SUBAPPLICATION Uebung_122_AX (* Übung zu ISOBUS Name *)
  (* Standard: 61499-2; Description: Copyright (c) 2023 Meisterschulen am Ostbahnhof This program and the accompanying materials are made available under the terms of the Eclipse Public License 2.0 which is available at https://www.eclipse.org/legal/epl-2.0/ SPDX-License-Identifier: EPL-2.0 *)
  (* Version 1.0, 2023-10-23, Franz Höpfinger, Meisterschulen am Ostbahnhof, initial API and implementation and/or initial documentation *)
  PACKAGE Uebungen;
  IMPORT Uebungen::const::Uebung_120_129::Filter::ADD_ALL_PASS;
  IMPORT Uebungen::const::Uebung_120_129::Filter::FLT_ALL_PASS;
  IMPORT isobus::pgn::ISOUSERHOME_e::network;
  IMPORT isobus::pgn::ISO_CAN_NODE::NODE1;
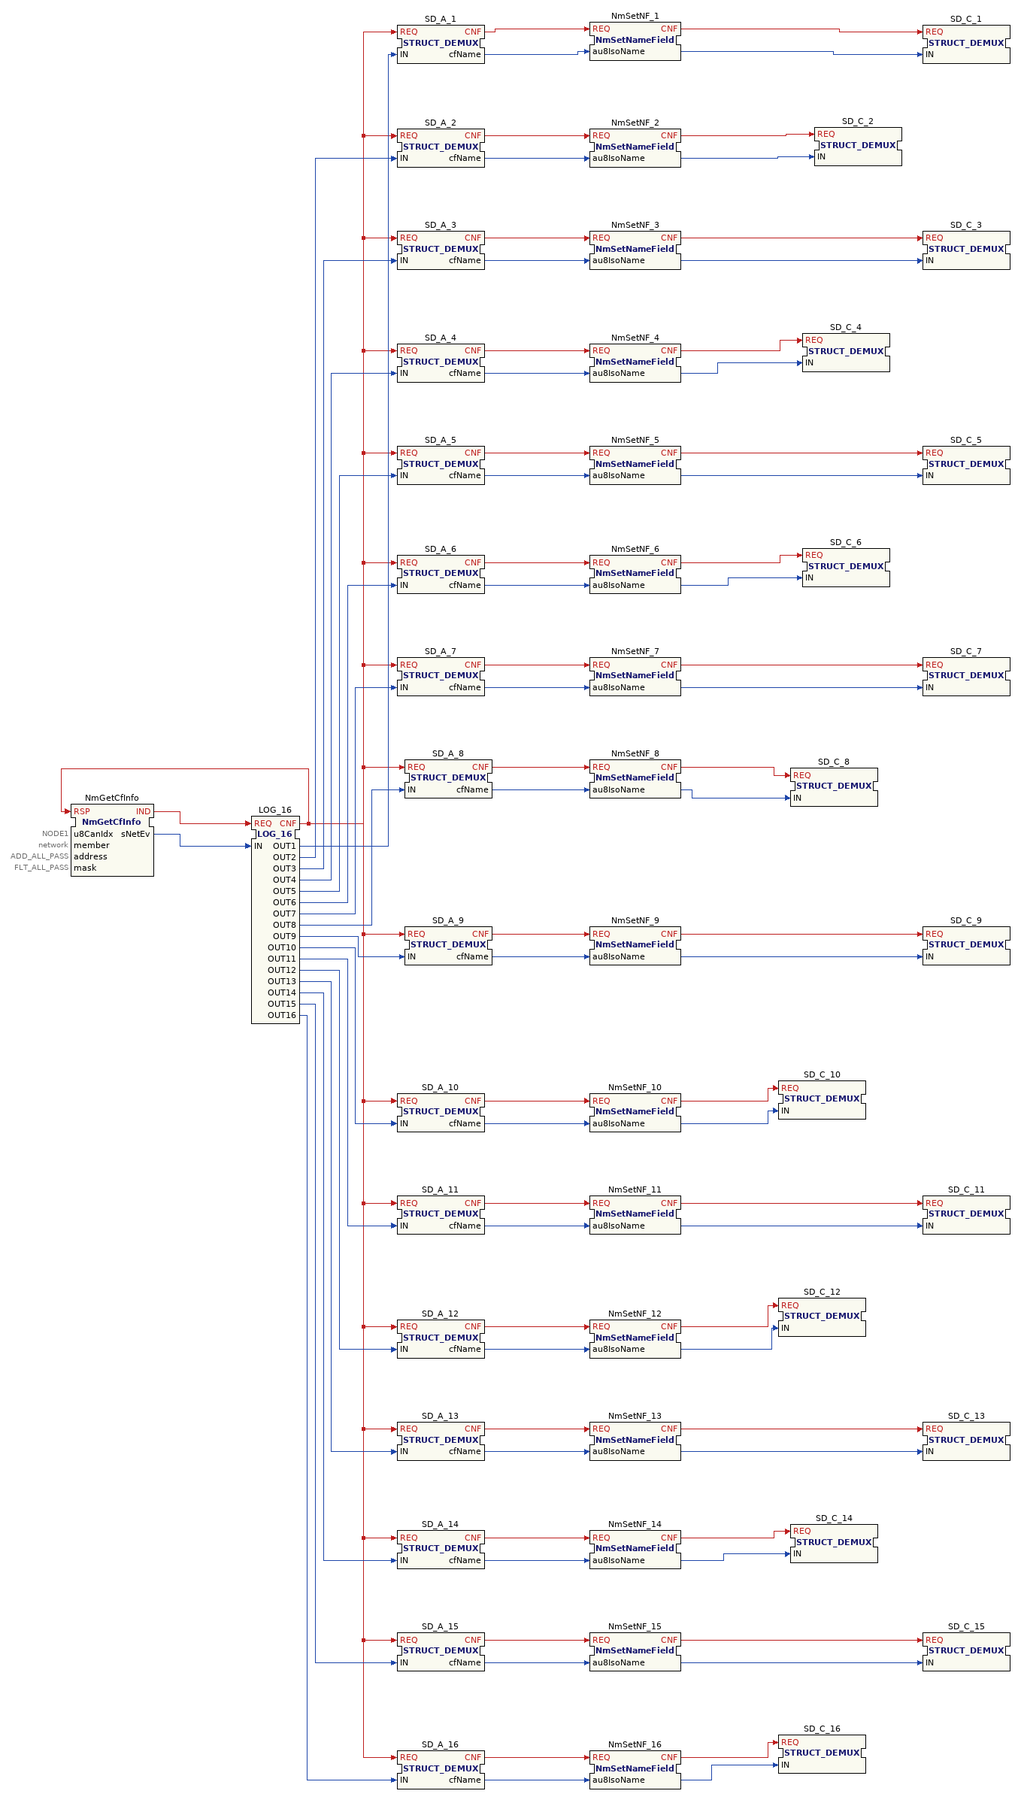
  FBS
    NmGetCfInfo : isobus::pgn::NmGetCfInfo(u8CanIdx := NODE1, member := network, address := ADD_ALL_PASS, mask := FLT_ALL_PASS);
    LOG_16 : logiBUS::utils::logging::LOG_16;
    SD_A_1 : eclipse4diac::convert::STRUCT_DEMUX; {SET_ATTRIBUTE(StructuredType, isobus::pgn::ISONETEVENT_T)}
    SD_A_2 : eclipse4diac::convert::STRUCT_DEMUX; {SET_ATTRIBUTE(StructuredType, isobus::pgn::ISONETEVENT_T)}
    SD_A_3 : eclipse4diac::convert::STRUCT_DEMUX; {SET_ATTRIBUTE(StructuredType, isobus::pgn::ISONETEVENT_T)}
    SD_A_4 : eclipse4diac::convert::STRUCT_DEMUX; {SET_ATTRIBUTE(StructuredType, isobus::pgn::ISONETEVENT_T)}
    SD_A_5 : eclipse4diac::convert::STRUCT_DEMUX; {SET_ATTRIBUTE(StructuredType, isobus::pgn::ISONETEVENT_T)}
    SD_A_6 : eclipse4diac::convert::STRUCT_DEMUX; {SET_ATTRIBUTE(StructuredType, isobus::pgn::ISONETEVENT_T)}
    SD_A_7 : eclipse4diac::convert::STRUCT_DEMUX; {SET_ATTRIBUTE(StructuredType, isobus::pgn::ISONETEVENT_T)}
    SD_A_8 : eclipse4diac::convert::STRUCT_DEMUX; {SET_ATTRIBUTE(StructuredType, isobus::pgn::ISONETEVENT_T)}
    SD_A_9 : eclipse4diac::convert::STRUCT_DEMUX; {SET_ATTRIBUTE(StructuredType, isobus::pgn::ISONETEVENT_T)}
    SD_A_10 : eclipse4diac::convert::STRUCT_DEMUX; {SET_ATTRIBUTE(StructuredType, isobus::pgn::ISONETEVENT_T)}
    SD_A_11 : eclipse4diac::convert::STRUCT_DEMUX; {SET_ATTRIBUTE(StructuredType, isobus::pgn::ISONETEVENT_T)}
    SD_A_12 : eclipse4diac::convert::STRUCT_DEMUX; {SET_ATTRIBUTE(StructuredType, isobus::pgn::ISONETEVENT_T)}
    SD_A_13 : eclipse4diac::convert::STRUCT_DEMUX; {SET_ATTRIBUTE(StructuredType, isobus::pgn::ISONETEVENT_T)}
    SD_A_14 : eclipse4diac::convert::STRUCT_DEMUX; {SET_ATTRIBUTE(StructuredType, isobus::pgn::ISONETEVENT_T)}
    SD_A_15 : eclipse4diac::convert::STRUCT_DEMUX; {SET_ATTRIBUTE(StructuredType, isobus::pgn::ISONETEVENT_T)}
    SD_A_16 : eclipse4diac::convert::STRUCT_DEMUX; {SET_ATTRIBUTE(StructuredType, isobus::pgn::ISONETEVENT_T)}
    NmSetNF_1 : isobus::pgn::NmSetNameField;
    NmSetNF_2 : isobus::pgn::NmSetNameField;
    NmSetNF_3 : isobus::pgn::NmSetNameField;
    NmSetNF_4 : isobus::pgn::NmSetNameField;
    NmSetNF_5 : isobus::pgn::NmSetNameField;
    NmSetNF_6 : isobus::pgn::NmSetNameField;
    NmSetNF_7 : isobus::pgn::NmSetNameField;
    NmSetNF_8 : isobus::pgn::NmSetNameField;
    NmSetNF_9 : isobus::pgn::NmSetNameField;
    NmSetNF_10 : isobus::pgn::NmSetNameField;
    NmSetNF_11 : isobus::pgn::NmSetNameField;
    NmSetNF_12 : isobus::pgn::NmSetNameField;
    NmSetNF_13 : isobus::pgn::NmSetNameField;
    NmSetNF_14 : isobus::pgn::NmSetNameField;
    NmSetNF_15 : isobus::pgn::NmSetNameField;
    NmSetNF_16 : isobus::pgn::NmSetNameField;
    SD_C_1 : eclipse4diac::convert::STRUCT_DEMUX; {SET_ATTRIBUTE(StructuredType, isobus::pgn::NAMEFIELD_T)}
    SD_C_2 : eclipse4diac::convert::STRUCT_DEMUX; {SET_ATTRIBUTE(StructuredType, isobus::pgn::NAMEFIELD_T)}
    SD_C_3 : eclipse4diac::convert::STRUCT_DEMUX; {SET_ATTRIBUTE(StructuredType, isobus::pgn::NAMEFIELD_T)}
    SD_C_4 : eclipse4diac::convert::STRUCT_DEMUX; {SET_ATTRIBUTE(StructuredType, isobus::pgn::NAMEFIELD_T)}
    SD_C_5 : eclipse4diac::convert::STRUCT_DEMUX; {SET_ATTRIBUTE(StructuredType, isobus::pgn::NAMEFIELD_T)}
    SD_C_6 : eclipse4diac::convert::STRUCT_DEMUX; {SET_ATTRIBUTE(StructuredType, isobus::pgn::NAMEFIELD_T)}
    SD_C_7 : eclipse4diac::convert::STRUCT_DEMUX; {SET_ATTRIBUTE(StructuredType, isobus::pgn::NAMEFIELD_T)}
    SD_C_8 : eclipse4diac::convert::STRUCT_DEMUX; {SET_ATTRIBUTE(StructuredType, isobus::pgn::NAMEFIELD_T)}
    SD_C_9 : eclipse4diac::convert::STRUCT_DEMUX; {SET_ATTRIBUTE(StructuredType, isobus::pgn::NAMEFIELD_T)}
    SD_C_10 : eclipse4diac::convert::STRUCT_DEMUX; {SET_ATTRIBUTE(StructuredType, isobus::pgn::NAMEFIELD_T)}
    SD_C_11 : eclipse4diac::convert::STRUCT_DEMUX; {SET_ATTRIBUTE(StructuredType, isobus::pgn::NAMEFIELD_T)}
    SD_C_12 : eclipse4diac::convert::STRUCT_DEMUX; {SET_ATTRIBUTE(StructuredType, isobus::pgn::NAMEFIELD_T)}
    SD_C_13 : eclipse4diac::convert::STRUCT_DEMUX; {SET_ATTRIBUTE(StructuredType, isobus::pgn::NAMEFIELD_T)}
    SD_C_14 : eclipse4diac::convert::STRUCT_DEMUX; {SET_ATTRIBUTE(StructuredType, isobus::pgn::NAMEFIELD_T)}
    SD_C_15 : eclipse4diac::convert::STRUCT_DEMUX; {SET_ATTRIBUTE(StructuredType, isobus::pgn::NAMEFIELD_T)}
    SD_C_16 : eclipse4diac::convert::STRUCT_DEMUX; {SET_ATTRIBUTE(StructuredType, isobus::pgn::NAMEFIELD_T)}
  END_FBS
  EVENT_CONNECTIONS
    NmGetCfInfo.IND TO LOG_16.REQ;
    LOG_16.CNF TO SD_A_1.REQ;
    LOG_16.CNF TO SD_A_2.REQ;
    LOG_16.CNF TO SD_A_3.REQ;
    LOG_16.CNF TO SD_A_4.REQ;
    LOG_16.CNF TO SD_A_5.REQ;
    LOG_16.CNF TO SD_A_6.REQ;
    LOG_16.CNF TO SD_A_7.REQ;
    LOG_16.CNF TO SD_A_8.REQ;
    LOG_16.CNF TO SD_A_9.REQ;
    LOG_16.CNF TO SD_A_10.REQ;
    LOG_16.CNF TO SD_A_11.REQ;
    LOG_16.CNF TO SD_A_12.REQ;
    LOG_16.CNF TO SD_A_13.REQ;
    LOG_16.CNF TO SD_A_14.REQ;
    LOG_16.CNF TO SD_A_15.REQ;
    LOG_16.CNF TO SD_A_16.REQ;
    SD_A_1.CNF TO NmSetNF_1.REQ;
    NmSetNF_1.CNF TO SD_C_1.REQ;
    SD_A_2.CNF TO NmSetNF_2.REQ;
    NmSetNF_2.CNF TO SD_C_2.REQ;
    SD_A_3.CNF TO NmSetNF_3.REQ;
    NmSetNF_3.CNF TO SD_C_3.REQ;
    SD_A_4.CNF TO NmSetNF_4.REQ;
    NmSetNF_4.CNF TO SD_C_4.REQ;
    SD_A_5.CNF TO NmSetNF_5.REQ;
    NmSetNF_5.CNF TO SD_C_5.REQ;
    SD_A_6.CNF TO NmSetNF_6.REQ;
    NmSetNF_6.CNF TO SD_C_6.REQ;
    SD_A_7.CNF TO NmSetNF_7.REQ;
    NmSetNF_7.CNF TO SD_C_7.REQ;
    SD_A_8.CNF TO NmSetNF_8.REQ;
    NmSetNF_8.CNF TO SD_C_8.REQ;
    SD_A_9.CNF TO NmSetNF_9.REQ;
    NmSetNF_9.CNF TO SD_C_9.REQ;
    SD_A_10.CNF TO NmSetNF_10.REQ;
    NmSetNF_10.CNF TO SD_C_10.REQ;
    SD_A_11.CNF TO NmSetNF_11.REQ;
    NmSetNF_11.CNF TO SD_C_11.REQ;
    SD_A_12.CNF TO NmSetNF_12.REQ;
    NmSetNF_12.CNF TO SD_C_12.REQ;
    SD_A_13.CNF TO NmSetNF_13.REQ;
    NmSetNF_13.CNF TO SD_C_13.REQ;
    SD_A_14.CNF TO NmSetNF_14.REQ;
    NmSetNF_14.CNF TO SD_C_14.REQ;
    SD_A_15.CNF TO NmSetNF_15.REQ;
    NmSetNF_15.CNF TO SD_C_15.REQ;
    SD_A_16.CNF TO NmSetNF_16.REQ;
    NmSetNF_16.CNF TO SD_C_16.REQ;
    LOG_16.CNF TO NmGetCfInfo.RSP;
  END_CONNECTIONS
  DATA_CONNECTIONS
    NmGetCfInfo.sNetEv TO LOG_16.IN;
    LOG_16.OUT1 TO SD_A_1.IN;
    LOG_16.OUT2 TO SD_A_2.IN;
    LOG_16.OUT3 TO SD_A_3.IN;
    LOG_16.OUT4 TO SD_A_4.IN;
    LOG_16.OUT5 TO SD_A_5.IN;
    LOG_16.OUT6 TO SD_A_6.IN;
    LOG_16.OUT7 TO SD_A_7.IN;
    LOG_16.OUT8 TO SD_A_8.IN;
    LOG_16.OUT9 TO SD_A_9.IN;
    LOG_16.OUT10 TO SD_A_10.IN;
    LOG_16.OUT11 TO SD_A_11.IN;
    LOG_16.OUT12 TO SD_A_12.IN;
    LOG_16.OUT13 TO SD_A_13.IN;
    LOG_16.OUT14 TO SD_A_14.IN;
    LOG_16.OUT15 TO SD_A_15.IN;
    LOG_16.OUT16 TO SD_A_16.IN;
    SD_A_1.cfName TO NmSetNF_1.au8IsoName;
    SD_A_2.cfName TO NmSetNF_2.au8IsoName;
    SD_A_3.cfName TO NmSetNF_3.au8IsoName;
    SD_A_4.cfName TO NmSetNF_4.au8IsoName;
    SD_A_5.cfName TO NmSetNF_5.au8IsoName;
    SD_A_6.cfName TO NmSetNF_6.au8IsoName;
    SD_A_7.cfName TO NmSetNF_7.au8IsoName;
    SD_A_8.cfName TO NmSetNF_8.au8IsoName;
    SD_A_9.cfName TO NmSetNF_9.au8IsoName;
    SD_A_10.cfName TO NmSetNF_10.au8IsoName;
    SD_A_11.cfName TO NmSetNF_11.au8IsoName;
    SD_A_12.cfName TO NmSetNF_12.au8IsoName;
    SD_A_13.cfName TO NmSetNF_13.au8IsoName;
    SD_A_14.cfName TO NmSetNF_14.au8IsoName;
    SD_A_15.cfName TO NmSetNF_15.au8IsoName;
    SD_A_16.cfName TO NmSetNF_16.au8IsoName;
    NmSetNF_1. TO SD_C_1.IN;
    NmSetNF_2. TO SD_C_2.IN;
    NmSetNF_3. TO SD_C_3.IN;
    NmSetNF_4. TO SD_C_4.IN;
    NmSetNF_5. TO SD_C_5.IN;
    NmSetNF_6. TO SD_C_6.IN;
    NmSetNF_7. TO SD_C_7.IN;
    NmSetNF_8. TO SD_C_8.IN;
    NmSetNF_9. TO SD_C_9.IN;
    NmSetNF_10. TO SD_C_10.IN;
    NmSetNF_11. TO SD_C_11.IN;
    NmSetNF_12. TO SD_C_12.IN;
    NmSetNF_13. TO SD_C_13.IN;
    NmSetNF_14. TO SD_C_14.IN;
    NmSetNF_15. TO SD_C_15.IN;
    NmSetNF_16. TO SD_C_16.IN;
  END_CONNECTIONS
END_SUBAPPLICATION
